// Mitsubishi GX Works2 project: RETENTIVE_TIMER   PLC: Q03UDV

PROGRAM MAIN
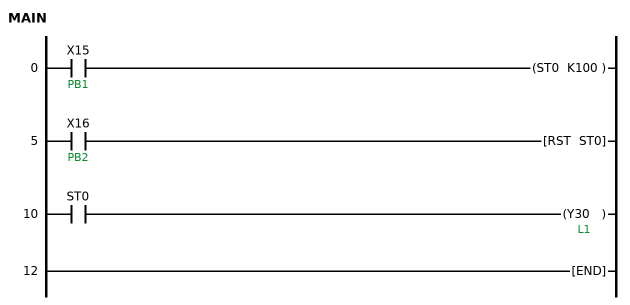
0     LD      X15  ; PB1
      OUT     ST0 K100
5     LD      X16  ; PB2
      RST     ST0
10    LD      ST0
      OUT     Y30  ; L1
12    END
END_PROGRAM

// device comments not shown above
X17  ; PB3
X18  ; PB4
X19  ; PB5
X1A  ; PB6
Y31  ; L2
Y32  ; L3
Y33  ; L4
Y34  ; L5
Y35  ; L6
Y36  ; L7
Y37  ; L8
T0  ; 타이머1
T1  ; 타이머2
T2  ; 타이머3
T3  ; 타이머4
T4  ; 타이머5
T5  ; 타이머6
T6  ; 타이머7
T7  ; 타이머8
T8  ; 타이머 9
T9  ; 타이머10
T10  ; 타이머11
T11  ; 타이머12
